FUNCTION_BLOCK FB_Cinta EXTENDS FB_Module
VAR_INPUT
	situar: BOOL;
	transportar: BOOL;
END_VAR
VAR_OUTPUT
END_VAR
VAR
	fbController: FB_Cinta_SFC;
	(*Sensores*)
	pp    : dvSensor;
	(*Actuadores*)
	R_1   : dvActuator := (tm:=tm);
	S_1   : dvActuator := (tm:=tm);
	RUN   : dvActuator := (tm:=tm);
	REV   : dvActuator := (tm:=tm);
	
END_VAR

METHOD ModuleControlFlow : BOOL
fbController(	
	tm := tm, IC:=IC, Execute:=Execute, Ack:=Ack,
	Ready=>Ready, Done=>Done, Failure=>Failure);
END_METHOD

END_FUNCTION_BLOCK

(* stored: Version 1.1.0.1, ProductVersion 3.1.4024.6
   POU FB_Cinta: Id {f4de692b-96c6-493e-9b33-3a90e20acfad}, SpecialFunc None
   Method ModuleControlFlow: Id {8ef223d1-a933-4fe3-87e8-40d9ed750433} *)
